// TIA Portal V17 export
// export: Created 2023-04-07T13:41:57.6288938Z, ExportSetting WithDefaults, DisplayName Totally Integrated Automation Portal, DisplayVersion V17 Update 4, DisplayName TIA Portal Openness, DisplayVersion V17 Update 4, DisplayName TIA Portal Version Control Interface, DisplayVersion V17, DisplayName STEP 7 Professional, DisplayVersion V17 Update 4, DisplayName STEP 7 Safety, DisplayVersion V17, DisplayName WinCC Professional, DisplayVersion V17 Update 4
FUNCTION "Digital Output" : Void   // FC5, LAD
{ S7_Optimized_Access := 'TRUE' }
VERSION : 0.1
// stored: AutoNumber false, IsIECCheckEnabled false, SetENOAutomatically false, UDAEnableTagReadback false
BEGIN

REGION Network 1: Digital Output 1
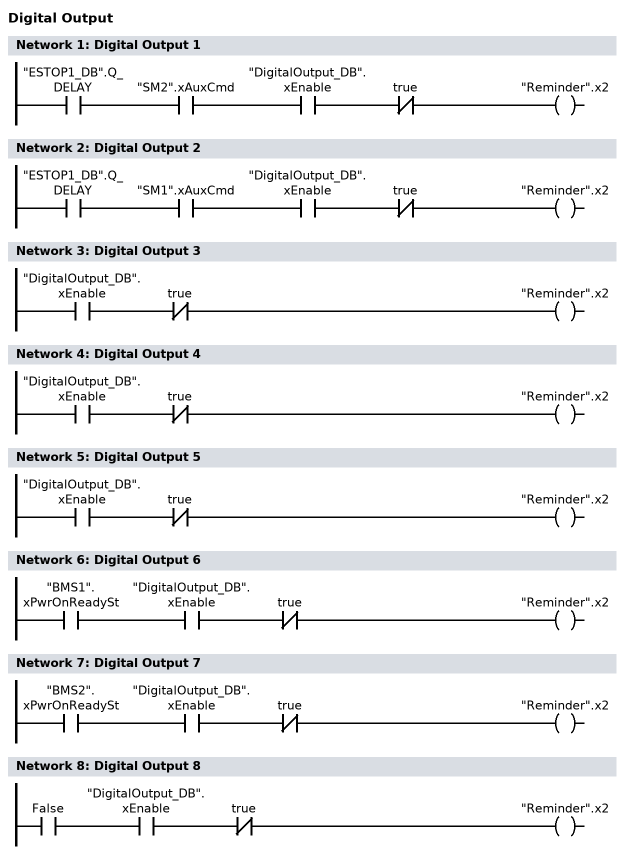
   RUNG wire#powerrail
      Contact( "ESTOP1_DB".Q_DELAY )
      Contact( "SM2".xAuxCmd )
      Contact( "DigitalOutput_DB".xEnable )
      I_Contact( true )
      Coil( "Reminder".x2 )
   END_RUNG
   // the same network as SCL:
   "Reminder".x2 := "ESTOP1_DB".Q_DELAY AND "SM2".xAuxCmd AND "DigitalOutput_DB".xEnable AND NOT true;
END_REGION

REGION Network 2: Digital Output 2
   RUNG wire#powerrail
      Contact( "ESTOP1_DB".Q_DELAY )
      Contact( "SM1".xAuxCmd )
      Contact( "DigitalOutput_DB".xEnable )
      I_Contact( true )
      Coil( "Reminder".x2 )
   END_RUNG
   // the same network as SCL:
   "Reminder".x2 := "ESTOP1_DB".Q_DELAY AND "SM1".xAuxCmd AND "DigitalOutput_DB".xEnable AND NOT true;
END_REGION

REGION Network 3: Digital Output 3
   RUNG wire#powerrail
      Contact( "DigitalOutput_DB".xEnable )
      I_Contact( true )
      Coil( "Reminder".x2 )
   END_RUNG
   // the same network as SCL:
   "Reminder".x2 := "DigitalOutput_DB".xEnable AND NOT true;
END_REGION

REGION Network 4: Digital Output 4
   RUNG wire#powerrail
      Contact( "DigitalOutput_DB".xEnable )
      I_Contact( true )
      Coil( "Reminder".x2 )
   END_RUNG
   // the same network as SCL:
   "Reminder".x2 := "DigitalOutput_DB".xEnable AND NOT true;
END_REGION

REGION Network 5: Digital Output 5
   RUNG wire#powerrail
      Contact( "DigitalOutput_DB".xEnable )
      I_Contact( true )
      Coil( "Reminder".x2 )
   END_RUNG
   // the same network as SCL:
   "Reminder".x2 := "DigitalOutput_DB".xEnable AND NOT true;
END_REGION

REGION Network 6: Digital Output 6
   RUNG wire#powerrail
      Contact( "BMS1".xPwrOnReadySt )
      Contact( "DigitalOutput_DB".xEnable )
      I_Contact( true )
      Coil( "Reminder".x2 )
   END_RUNG
   // the same network as SCL:
   "Reminder".x2 := "BMS1".xPwrOnReadySt AND "DigitalOutput_DB".xEnable AND NOT true;
END_REGION

REGION Network 7: Digital Output 7
   RUNG wire#powerrail
      Contact( "BMS2".xPwrOnReadySt )
      Contact( "DigitalOutput_DB".xEnable )
      I_Contact( true )
      Coil( "Reminder".x2 )
   END_RUNG
   // the same network as SCL:
   "Reminder".x2 := "BMS2".xPwrOnReadySt AND "DigitalOutput_DB".xEnable AND NOT true;
END_REGION

REGION Network 8: Digital Output 8
   RUNG wire#powerrail
      Contact( False )
      Contact( "DigitalOutput_DB".xEnable )
      I_Contact( true )
      Coil( "Reminder".x2 )
   END_RUNG
   // the same network as SCL:
   "Reminder".x2 := False AND "DigitalOutput_DB".xEnable AND NOT true;
END_REGION
END_FUNCTION
